// TIA Portal V16 export
// export: Created 2022-07-21T09:35:16.0398925Z, ExportSetting WithDefaults, DisplayName Totally Integrated Automation Portal, DisplayVersion V16 Update 4, DisplayName TIA Portal Version Control Interface, DisplayVersion V16 Update 2, DisplayName TIA Portal Openness, DisplayVersion V16 Update 4, DisplayName SINAMICS Startdrive Advanced, DisplayVersion V16 Update 5, DisplayName SINAMICS Startdrive G130, G150, S120, S150, SINAMICS MV, S210, DisplayVersion V16 Update 5, DisplayName SINAMICS Startdrive G110M, G120, G120C, G120D, G120P, G115D, DisplayVersion V16 Update 5, DisplayName STEP 7 Professional, DisplayVersion V16 Update 4, DisplayName STEP 7 Safety, DisplayVersion V16, DisplayName WinCC Advanced, DisplayVersion V16 Update 4
FUNCTION_BLOCK "fbMessageHandlingDelayed"   // FB18, LAD
TITLE = Error handling / Obsługa błędów
{ S7_Optimized_Access := 'TRUE' }
VERSION : 0.1
// stored: AutoNumber true, IsIECCheckEnabled true, IsRetainMemResEnabled false, MemoryReserve 100, SetENOAutomatically false, UDAEnableTagReadback false
   VAR_INPUT
      inEnable { ExternalAccessible := 'False'; ExternalVisible := 'False'; ExternalWritable := 'False'} : Bool;   // Zezwolenie / Enable
      inFbSignalOk { ExternalAccessible := 'False'; ExternalVisible := 'False'; ExternalWritable := 'False'} : Bool;   // Sygnał ok / Signal ok
      inResetMessages { ExternalAccessible := 'False'; ExternalVisible := 'False'; ExternalWritable := 'False'} : Bool;   // Reset błędu / Reset error
      inDelaySignalOn { ExternalAccessible := 'False'; ExternalVisible := 'False'; ExternalWritable := 'False'} : Time;   // Opóźnienie ustawienia sygnału wejściowego / delay input signal set
      inDelaySignalOff { ExternalAccessible := 'False'; ExternalVisible := 'False'; ExternalWritable := 'False'} : Time;   // Opóźnienie wyłączenia sygnału wejsciowego / delay input signal reset
   END_VAR
   VAR_OUTPUT
      ouMessage { ExternalAccessible := 'False'; ExternalVisible := 'False'; ExternalWritable := 'False'} : Bool;   // Wygenerowany błąd / Generated error
   END_VAR
   VAR
      sTonDelaySignalOn { ExternalAccessible := 'False'; ExternalVisible := 'False'; ExternalWritable := 'False'; S7_SetPoint := 'True'} : IEC_TIMER;
      sTonDelaySignalOff { ExternalAccessible := 'False'; ExternalVisible := 'False'; ExternalWritable := 'False'; S7_SetPoint := 'True'} : IEC_TIMER;
      sSignalOk { ExternalAccessible := 'False'; ExternalVisible := 'False'; ExternalWritable := 'False'} : Bool;
   END_VAR
BEGIN

REGION Network 1: On delay / Opóznienie sygnału załącz
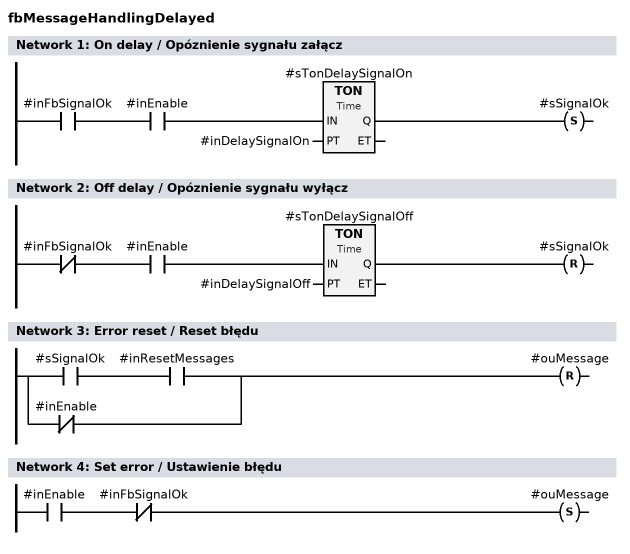
   RUNG wire#powerrail
      Contact( #inFbSignalOk )
      Contact( #inEnable )
      { S7_Templates := "time_type := Time" } #sTonDelaySignalOn.TON(pt := #inDelaySignalOn, et =>)
      S_Coil( #sSignalOk )
   END_RUNG
   // the same network as SCL:
   #sTonDelaySignalOn.TON(IN := #inFbSignalOk AND #inEnable, PT := #inDelaySignalOn);
   IF #sTonDelaySignalOn.Q THEN #sSignalOk := TRUE; END_IF;
END_REGION

REGION Network 2: Off delay / Opóznienie sygnału wyłącz
   RUNG wire#powerrail
      I_Contact( #inFbSignalOk )
      Contact( #inEnable )
      { S7_Templates := "time_type := Time" } #sTonDelaySignalOff.TON(pt := #inDelaySignalOff, et =>)
      R_Coil( #sSignalOk )
   END_RUNG
   // the same network as SCL:
   #sTonDelaySignalOff.TON(IN := NOT #inFbSignalOk AND #inEnable, PT := #inDelaySignalOff);
   IF #sTonDelaySignalOff.Q THEN #sSignalOk := FALSE; END_IF;
END_REGION

REGION Network 3: Error reset / Reset błędu
   RUNG wire#powerrail
      Contact( #sSignalOk )
      Contact( #inResetMessages )
      wire#w1
      R_Coil( #ouMessage )
   END_RUNG
   RUNG wire#powerrail
      I_Contact( #inEnable )
   END_RUNG wire#w1
   // the same network as SCL:
   IF (#sSignalOk AND #inResetMessages) OR NOT #inEnable THEN #ouMessage := FALSE; END_IF;
END_REGION

REGION Network 4: Set error / Ustawienie błędu
   RUNG wire#powerrail
      Contact( #inEnable )
      I_Contact( #inFbSignalOk )
      S_Coil( #ouMessage )
   END_RUNG
   // the same network as SCL:
   IF #inEnable AND NOT #inFbSignalOk THEN #ouMessage := TRUE; END_IF;
END_REGION
END_FUNCTION_BLOCK
